// TIA Portal V18 export
// export: Created 2026-06-22T11:43:40.4217629Z, ExportSetting WithDefaults, DisplayName Totally Integrated Automation Portal, DisplayVersion V18, DisplayName TIA Portal Openness, DisplayVersion V18, DisplayName TIA Portal Version Control Interface, DisplayVersion V18, DisplayName STEP 7 Professional, DisplayVersion V18, DisplayName STEP 7 Safety, DisplayVersion V18, DisplayName WinCC Professional, DisplayVersion V18
Screen "Man Tong Quan"  1440x900, Number=3
  ScreenLayer 
    GraphicView "Graphic view_1" at 0,0 size 1440x900  Picture=Thiết kế chưa có tên (2)_1
    GraphicIOField "Graphic I/O field_9" at 430,521 size 275x288  Mode=InOutput, OnValue=1, PictureList=GL_BonChua_MucDich
      ProcessValue := HMI_Anim_BonChua1_MucDich
    GraphicIOField "Graphic I/O field_10" at 154,90 size 233x295  Mode=InOutput, OnValue=1, PictureList=GL_BonTron_MucDich
      ProcessValue := HMI_Anim_Bon1_MucDich
    GraphicIOField "Graphic I/O field_2" at 904,517 size 275x288  Mode=InOutput, OnValue=1, PictureList=GL_BonChua_MucDich
      ProcessValue := HMI_Anim_BonChua2_MucDich
    GraphicIOField "Graphic I/O field_3" at 486,90 size 233x295  Mode=InOutput, OnValue=1, PictureList=GL_BonTron_MucDich
      ProcessValue := HMI_Anim_Bon2_MucDich
    GraphicIOField "Graphic I/O field_4" at 811,89 size 233x295  Mode=InOutput, OnValue=1, PictureList=GL_BonTron_MucDich
      ProcessValue := HMI_Anim_Bon4_MucDich
    GraphicIOField "Graphic I/O field_6" at 1160,89 size 233x295  Mode=InOutput, OnValue=1, PictureList=GL_BonTron_MucDich
      ProcessValue := HMI_Anim_Bon3_MucDich
    GraphicView "Graphic view_3" at 201,61 size 11x113  Picture=Graphic_24
    GraphicIOField "Graphic I/O field_5" at 189,70 size 51x78  Mode=InOutput, OnValue=1, PictureList=GL_Van_NamDoc
      ProcessValue := V3230_Nuoc_Bon1_M
    GraphicView "Graphic view_2" at 544,60 size 11x113  Picture=Graphic_24
    GraphicIOField "Graphic I/O field_12" at 533,70 size 51x78  Mode=InOutput, OnValue=1, PictureList=GL_Van_NamDoc
      ProcessValue := V3235_Nuoc_Bon2_M
    GraphicView "Graphic view_4" at 869,59 size 11x113  Picture=Graphic_24
    GraphicIOField "Graphic I/O field_13" at 860,69 size 51x78  Mode=InOutput, OnValue=1, PictureList=GL_Van_NamDoc
      ProcessValue := V3245_Nuoc_Bon4_M
    GraphicView "Graphic view_5" at 1204,58 size 11x117  Picture=Graphic_24
    GraphicIOField "Graphic I/O field_14" at 1193,67 size 51x78  Mode=InOutput, OnValue=1, PictureList=GL_Van_NamDoc
      ProcessValue := V3240_Nuoc_Bon3_M
    GraphicView "Graphic view_6" at 229,330 size 11x172  Picture=Graphic_24
    GraphicIOField "Graphic I/O field_11" at 220,429 size 51x78  Mode=InOutput, OnValue=1, PictureList=GL_Van_NamDoc
      ProcessValue := V3233_Xa_Bon1_M
    GraphicIOField "Graphic I/O field_8" at 220,339 size 51x78  Mode=InOutput, OnValue=1, PictureList=GL_Van_NamDoc
      ProcessValue := V3232_Xa_Bon1_M
    GraphicView "Graphic view_7" at 568,331 size 11x211  Picture=Graphic_24
    GraphicView "Graphic view_8" at 869,328 size 11x164  Picture=Graphic_24
    GraphicView "Graphic view_9" at 1224,328 size 11x164  Picture=Graphic_24
    GraphicIOField "Graphic I/O field_15" at 556,341 size 51x78  Mode=InOutput, OnValue=1, PictureList=GL_Van_NamDoc
      ProcessValue := V3237_Xa_Bon2_M
    GraphicIOField "Graphic I/O field_16" at 558,417 size 51x78  Mode=InOutput, OnValue=1, PictureList=GL_Van_NamDoc
      ProcessValue := V3238_Xa_Bon2_M
    GraphicIOField "Graphic I/O field_18" at 857,346 size 51x78  Mode=InOutput, OnValue=1, PictureList=GL_Van_NamDoc
      ProcessValue := V3247_Xa_Bon4_M
    GraphicIOField "Graphic I/O field_20" at 857,412 size 51x78  Mode=InOutput, OnValue=1, PictureList=GL_Van_NamDoc
      ProcessValue := V3248_Xa_Bon4_M
    GraphicIOField "Graphic I/O field_19" at 1214,347 size 51x78  Mode=InOutput, OnValue=1, PictureList=GL_Van_NamDoc
      ProcessValue := V3242_Xa_Bon3_M
    GraphicIOField "Graphic I/O field_21" at 1213,419 size 51x78  Mode=InOutput, OnValue=1, PictureList=GL_Van_NamDoc
      ProcessValue := V3243_Xa_Bon3_M
    GraphicView "Graphic view_10" at 223,500 size 25x5  Picture=Graphic_25
    GraphicView "Graphic view_11" at 1216,490 size 25x5  Picture=Graphic_25
    GraphicView "Graphic view_12" at 223,523 size 25x5  Picture=Graphic_25
    GraphicView "Graphic view_13" at 1216,515 size 25x5  Picture=Graphic_25
    GraphicView "Graphic view_14" at 252,501 size 5x26  Picture=Graphic_24
    GraphicView "Graphic view_15" at 1206,492 size 5x26  Picture=Graphic_24
    GraphicView "Graphic view_16" at 254,510 size 242x11  Picture=Graphic_25
    GraphicView "Graphic view_17" at 487,513 size 11x57  Picture=Graphic_24
    GraphicView "Graphic view_18" at 521,159 size 11x19  Picture=Graphic_24
    GraphicView "Graphic view_19" at 440,157 size 90x11  Picture=Graphic_25
    GraphicView "Graphic view_20" at 437,160 size 11x408  Picture=Graphic_24
    GraphicView "Graphic view_21" at 231,560 size 213x11  Picture=Graphic_25
    GraphicView "Graphic view_22" at 228,525 size 11x44  Picture=Graphic_24
    GraphicView "Graphic view_23" at 630,485 size 248x11  Picture=Graphic_25
    GraphicView "Graphic view_24" at 626,488 size 11x75  Picture=Graphic_24
    GraphicView "Graphic view_25" at 640,503 size 11x68  Picture=Graphic_24
    GraphicView "Graphic view_26" at 644,501 size 566x11  Picture=Graphic_25
    GraphicView "Graphic view_27" at 1224,517 size 11x51  Picture=Graphic_24
    GraphicView "Graphic view_28" at 1142,560 size 90x11  Picture=Graphic_25
    GraphicView "Graphic view_29" at 1139,99 size 11x469  Picture=Graphic_24
    GraphicView "Graphic view_30" at 1005,93 size 143x11  Picture=Graphic_25
    GraphicView "Graphic view_31" at 1000,95 size 11x86  Picture=Graphic_24
    GraphicView "Graphic view_32" at 564,755 size 11x103  Picture=Graphic_24
    GraphicIOField "Graphic I/O field_24" at 554,759 size 51x78  Mode=InOutput, OnValue=1, PictureList=GL_Van_NamDoc
      ProcessValue := V3331_Xa_BonChua1_M
    GraphicView "Graphic view_33" at 567,849 size 22x11  Picture=Graphic_25
    GraphicView "Graphic view_34" at 581,833 size 11x40  Picture=Graphic_24
    GraphicView "Graphic view_36" at 132,426 size 8x44  Picture=Graphic_28
    GraphicView "Graphic view_35" at 133,425 size 103x6  Picture=Graphic_29
    GraphicIOField "Graphic I/O field_7" at 133,396 size 83x47  Mode=InOutput, OnValue=1, PictureList=GL_Van_NamNgang
      ProcessValue := V3234_Xa_Bon1_M
    GraphicIOField "Graphic I/O field_33" at 282,542 size 60x42  Mode=InOutput, OnValue=1, PictureList=GL_Pump_ChuyenDich
      ProcessValue := Pump3264_Chuyen_Nhanh1_M
    GraphicView "Graphic view_38" at 371,61 size 2x119  Picture=Graphic_24
    GraphicView "Graphic view_40" at 352,178 size 22x2  Picture=Graphic_25
    GraphicView "Graphic view_39" at 361,99 size 21x47  Picture=Graphic_32
    GraphicView "Graphic view_41" at 125,453 size 21x47  Picture=Graphic_32
    GraphicView "Graphic view_37" at 341,167 size 28x25  Picture=Graphic_34
    GraphicView "Graphic view_42" at 473,422 size 103x6  Picture=Graphic_29
    GraphicIOField "Graphic I/O field_17" at 471,394 size 83x47  Mode=InOutput, OnValue=1, PictureList=GL_Van_NamNgang
      ProcessValue := V3239_Xa_Bon2_M
    GraphicView "Graphic view_43" at 472,423 size 8x44  Picture=Graphic_28
    GraphicView "Graphic view_44" at 466,451 size 21x47  Picture=Graphic_32
    GraphicView "Graphic view_45" at 872,415 size 108x6  Picture=Graphic_29
    GraphicIOField "Graphic I/O field_22" at 903,387 size 83x47  Mode=InOutput, OnValue=1, PictureList=GL_Van_NamNgang
      ProcessValue := V3249_Xa_Bon4_M
    GraphicView "Graphic view_46" at 976,415 size 8x35  Picture=Graphic_28
    GraphicView "Graphic view_47" at 970,434 size 21x47  Picture=Graphic_32
    GraphicView "Graphic view_48" at 1226,422 size 118x6  Picture=Graphic_29
    GraphicIOField "Graphic I/O field_23" at 1257,394 size 83x47  Mode=InOutput, OnValue=1, PictureList=GL_Van_NamNgang
      ProcessValue := V3244_Xa_Bon3_M
    GraphicView "Graphic view_49" at 1336,422 size 8x35  Picture=Graphic_28
    GraphicView "Graphic view_50" at 1331,441 size 21x47  Picture=Graphic_32
    GraphicView "Graphic view_51" at 709,59 size 2x119  Picture=Graphic_24
    GraphicView "Graphic view_52" at 1047,60 size 2x116  Picture=Graphic_24
    GraphicView "Graphic view_53" at 1387,60 size 2x114  Picture=Graphic_24
    GraphicView "Graphic view_54" at 700,102 size 21x47  Picture=Graphic_32
    GraphicView "Graphic view_55" at 1038,104 size 21x47  Picture=Graphic_32
    GraphicView "Graphic view_56" at 1378,106 size 21x47  Picture=Graphic_32
    GraphicView "Graphic view_57" at 689,177 size 22x2  Picture=Graphic_25
    GraphicView "Graphic view_58" at 1016,175 size 33x2  Picture=Graphic_25
    GraphicView "Graphic view_59" at 1366,173 size 22x2  Picture=Graphic_25
    GraphicView "Graphic view_60" at 672,166 size 28x25  Picture=Graphic_34
    GraphicView "Graphic view_61" at 1000,165 size 28x25  Picture=Graphic_34
    GraphicView "Graphic view_62" at 1347,162 size 28x25  Picture=Graphic_34
    GraphicView "Graphic view_63" at 584,865 size 16x11  Picture=Graphic_25
    GraphicView "Graphic view_64" at 584,830 size 159x11  Picture=Graphic_25
    GraphicView "Graphic view_65" at 598,858 size 5x26  Picture=Graphic_24
    GraphicView "Graphic view_66" at 603,858 size 5x26  Picture=Graphic_24
    GraphicView "Graphic view_67" at 605,866 size 68x11  Picture=Graphic_25
    GraphicIOField "Graphic I/O field_1" at 608,851 size 60x42  Mode=InOutput, OnValue=1, PictureList=GL_Pump_ChuyenDich
      ProcessValue := Pump3362_Xa_BonChua1_M
    GraphicView "Graphic view_68" at 668,858 size 5x26  Picture=Graphic_24
    GraphicView "Graphic view_69" at 674,858 size 5x26  Picture=Graphic_24
    GraphicView "Graphic view_70" at 675,866 size 13x11  Picture=Graphic_25
    GraphicView "Graphic view_71" at 682,513 size 11x361  Picture=Graphic_24
    GraphicIOField "Graphic I/O field_25" at 672,597 size 51x78  Mode=InOutput, OnValue=1, PictureList=GL_Van_NamDoc
      ProcessValue := V3333_DieuHuong_BonChua1_M
    GraphicView "Graphic view_72" at 684,510 size 376x11  Picture=Graphic_25
    GraphicView "Graphic view_73" at 1053,512 size 11x26  Picture=Graphic_24
    GraphicIOField "Graphic I/O field_34" at 587,792 size 90x71  Mode=InOutput, OnValue=1, PictureList=GL_Pump_TuanHoanLoc
      ProcessValue := Pump3361_LuanChuyen_BonChua1_M
    GraphicView "Graphic view_74" at 735,752 size 11x144  Picture=Graphic_24
    GraphicIOField "Graphic I/O field_27" at 725,829 size 51x78  Mode=InOutput, OnValue=1, PictureList=GL_Van_NamDoc
      ProcessValue := V3335_DieuHuong_BonChua1_M
    GraphicIOField "Graphic I/O field_26" at 725,757 size 51x78  Mode=InOutput, OnValue=1, PictureList=GL_Van_NamDoc
      ProcessValue := V3334_DieuHuong_BonChua1_M
    GraphicView "Graphic view_75" at 739,889 size 528x11  Picture=Graphic_25
    GraphicView "Graphic view_76" at 738,748 size 65x11  Picture=Graphic_25
    GraphicView "Graphic view_77" at 799,521 size 11x236  Picture=Graphic_24
    GraphicView "Graphic view_78" at 801,518 size 211x11  Picture=Graphic_25
    GraphicView "Graphic view_79" at 1005,520 size 11x38  Picture=Graphic_24
    GraphicView "Graphic view_80" at 469,833 size 103x6  Picture=Graphic_29
    GraphicView "Graphic view_81" at 467,834 size 8x44  Picture=Graphic_28
    GraphicView "Graphic view_82" at 461,854 size 21x47  Picture=Graphic_32
    GraphicIOField "Graphic I/O field_30" at 467,804 size 83x47  Mode=InOutput, OnValue=1, PictureList=GL_Van_NamNgang
      ProcessValue := V3332_Xa_BonChua1_M
    GraphicView "Graphic view_83" at 1040,751 size 11x75  Picture=Graphic_24
    GraphicIOField "Graphic I/O field_28" at 1030,754 size 51x78  Mode=InOutput, OnValue=1, PictureList=GL_Van_NamDoc
      ProcessValue := V3338_Xa_BonChua2_M
    GraphicView "Graphic view_84" at 1042,818 size 62x11  Picture=Graphic_25
    GraphicView "Graphic view_85" at 1100,802 size 11x40  Picture=Graphic_24
    GraphicView "Graphic view_86" at 1104,800 size 103x11  Picture=Graphic_25
    GraphicIOField "Graphic I/O field_35" at 1108,764 size 90x71  Mode=InOutput, OnValue=1, PictureList=GL_Pump_TuanHoanLoc
      ProcessValue := Pump3364_Filter_M
    GraphicView "Graphic view_87" at 1103,833 size 12x11  Picture=Graphic_25
    GraphicView "Graphic view_88" at 1112,825 size 5x26  Picture=Graphic_24
    GraphicView "Graphic view_89" at 1117,825 size 5x26  Picture=Graphic_24
    GraphicView "Graphic view_90" at 1118,833 size 72x11  Picture=Graphic_25
    GraphicIOField "Graphic I/O field_36" at 1123,820 size 60x42  Mode=InOutput, OnValue=1, PictureList=GL_Pump_ChuyenDich
      ProcessValue := Pump3365_Filter_M
    GraphicView "Graphic view_91" at 1186,825 size 5x26  Picture=Graphic_24
    GraphicView "Graphic view_92" at 1192,825 size 5x26  Picture=Graphic_24
    GraphicView "Graphic view_93" at 1195,833 size 13x11  Picture=Graphic_25
    GraphicView "Graphic view_94" at 1201,589 size 11x252  Picture=Graphic_24
    GraphicIOField "Graphic I/O field_29" at 1191,655 size 51x78  Mode=InOutput, OnValue=1, PictureList=GL_Van_NamDoc
      ProcessValue := V3340_Duong_Filter_M
    GraphicIOField "Graphic I/O field_37" at 1156,541 size 60x42  Mode=InOutput, OnValue=1, PictureList=GL_Pump_ChuyenDich
      ProcessValue := Pump3265_Chuyen_Nhanh2_M
    GraphicView "Graphic view_95" at 1204,587 size 150x11  Picture=Graphic_25
    GraphicView "Graphic view_96" at 1257,590 size 11x307  Picture=Graphic_24
    GraphicView "Graphic view_97" at 1345,589 size 11x192  Picture=Graphic_24
    GraphicView "Graphic view_98" at 1352,589 size 75x6  Picture=Graphic_29
    GraphicIOField "Graphic I/O field_32" at 1346,558 size 83x47  Mode=InOutput, OnValue=1, PictureList=GL_Van_NamNgang
      ProcessValue := V3341_Duong_Filter_M
    GraphicView "Graphic view_99" at 1420,591 size 8x35  Picture=Graphic_28
    GraphicView "Graphic view_100" at 1414,607 size 21x47  Picture=Graphic_32
    GraphicView "Graphic view_102" at 1368,50 size 41x72  Picture=Graphic_37
    GraphicView "Graphic view_103" at 1365,159 size 28x31  Picture=Graphic_38
    GraphicView "Graphic view_104" at 1027,50 size 41x72  Picture=Graphic_37
    GraphicView "Graphic view_105" at 690,50 size 41x72  Picture=Graphic_37
    GraphicView "Graphic view_106" at 352,50 size 41x72  Picture=Graphic_37
    GraphicView "Graphic view_107" at 352,121 size 41x74  Picture=Graphic_39
    GraphicView "Graphic view_108" at 691,121 size 41x74  Picture=Graphic_39
    GraphicView "Graphic view_109" at 1028,121 size 41x74  Picture=Graphic_39
    GraphicView "Graphic view_110" at 1368,119 size 41x74  Picture=Graphic_39
    GraphicView "Graphic view_101" at 1012,165 size 45x26  Picture=Graphic_40
    GraphicView "Graphic view_111" at 676,167 size 45x26  Picture=Graphic_40
    GraphicView "Graphic view_112" at 341,167 size 38x26  Picture=Graphic_40
    GraphicIOField "Graphic I/O field_38" at 123,84 size 292x298  Mode=Output, OnValue=1, PictureList=GL_Khuay_8Frame
      ProcessValue := HMI_Anim_Bon1_Frame
    GraphicIOField "Graphic I/O field_39" at 459,83 size 292x298  Mode=InOutput, OnValue=1, PictureList=GL_Khuay_8Frame
      ProcessValue := HMI_Anim_Bon2_Frame
    GraphicIOField "Graphic I/O field_40" at 782,86 size 292x298  Mode=InOutput, OnValue=1, PictureList=GL_Khuay_8Frame
      ProcessValue := HMI_Anim_Bon4_Frame
    GraphicIOField "Graphic I/O field_41" at 1130,89 size 292x298  Mode=InOutput, OnValue=1, PictureList=GL_Khuay_8Frame
      ProcessValue := HMI_Anim_Bon3_Frame
    GraphicView "Graphic view_113" at 1280,567 size 56x45  Picture=Graphic_44
    GraphicView "Graphic view_115" at 1338,606 size 28x43  Picture=Graphic_46
    GraphicView "Graphic view_114" at 1246,722 size 28x43  Picture=Graphic_46
    GraphicView "Graphic view_116" at 1340,714 size 33x47  Picture=Graphic_47
    GraphicView "Graphic view_117" at 1327,779 size 50x52  Picture=Graphic_48
    GraphicView "Graphic view_118" at 1341,815 size 21x47  Picture=Graphic_32
    GraphicView "Graphic view_119" at 1337,843 size 29x56  Picture=Graphic_49
    GraphicView "Graphic view_120" at 939,821 size 108x6  Picture=Graphic_29
    GraphicIOField "Graphic I/O field_31" at 930,792 size 83x47  Mode=InOutput, OnValue=1, PictureList=GL_Van_NamNgang
      ProcessValue := V3339_Xa_BonChua2_M
    GraphicView "Graphic view_121" at 934,821 size 8x44  Picture=Graphic_28
    GraphicView "Graphic view_122" at 929,842 size 21x47  Picture=Graphic_32
    IOField "I/O field_1" at 113,69 size 67x32  DataFormat=Decimal, FormatPattern=999999, Mode=InOutput
    GraphicView "Graphic view_123" at 775,636 size 55x48  Picture=Graphic_50
    IOField "I/O field_2" at 300,127 size 67x28  DataFormat=Decimal, FormatPattern=999999, Mode=InOutput
    TextField "AI_Lbl_Graphic I/O field_5" at 184,48 size 60x20  StyleItem=Text field, Text="<body><p>V32.30</p></body>"
    TextField "AI_Lbl_Graphic I/O field_12" at 528,48 size 60x20  StyleItem=Text field, Text="<body><p>V32.35</p></body>"
    TextField "AI_Lbl_Graphic I/O field_13" at 855,47 size 60x20  StyleItem=Text field, Text="<body><p>V32.45</p></body>"
    TextField "AI_Lbl_Graphic I/O field_14" at 1188,45 size 60x20  StyleItem=Text field, Text="<body><p>V32.40</p></body>"
    TextField "AI_Lbl_Graphic I/O field_8" at 215,317 size 60x20  StyleItem=Text field, Text="<body><p>V32.32</p></body>"
    TextField "AI_Lbl_Graphic I/O field_11" at 215,407 size 60x20  StyleItem=Text field, Text="<body><p>V32.33</p></body>"
    TextField "AI_Lbl_Graphic I/O field_7" at 144,445 size 60x20  StyleItem=Text field, Text="<body><p>V32.34</p></body>"
    TextField "AI_Lbl_Graphic I/O field_15" at 551,319 size 60x20  StyleItem=Text field, Text="<body><p>V32.37</p></body>"
    TextField "AI_Lbl_Graphic I/O field_16" at 553,395 size 60x20  StyleItem=Text field, Text="<body><p>V32.38</p></body>"
    TextField "AI_Lbl_Graphic I/O field_17" at 482,443 size 60x20  StyleItem=Text field, Text="<body><p>V32.39</p></body>"
    TextField "AI_Lbl_Graphic I/O field_18" at 852,324 size 60x20  StyleItem=Text field, Text="<body><p>V32.47</p></body>"
    TextField "AI_Lbl_Graphic I/O field_20" at 852,390 size 60x20  StyleItem=Text field, Text="<body><p>V32.48</p></body>"
    TextField "AI_Lbl_Graphic I/O field_22" at 914,436 size 60x20  StyleItem=Text field, Text="<body><p>V32.49</p></body>"
    TextField "AI_Lbl_Graphic I/O field_19" at 1209,325 size 60x20  StyleItem=Text field, Text="<body><p>V32.42</p></body>"
    TextField "AI_Lbl_Graphic I/O field_21" at 1208,397 size 60x20  StyleItem=Text field, Text="<body><p>V32.43</p></body>"
    TextField "AI_Lbl_Graphic I/O field_23" at 1268,443 size 60x20  StyleItem=Text field, Text="<body><p>V32.44</p></body>"
    TextField "AI_Lbl_Graphic I/O field_33" at 282,586 size 60x20  StyleItem=Text field, Text="<body><p>Pump 32.64</p></body>"
    TextField "AI_Lbl_Graphic I/O field_37" at 1156,585 size 60x20  StyleItem=Text field, Text="<body><p>Pump 32.69</p></body>"
    TextField "AI_Lbl_Graphic I/O field_24" at 549,737 size 60x20  StyleItem=Text field, Text="<body><p>V33.31</p></body>"
    TextField "AI_Lbl_Graphic I/O field_30" at 478,853 size 60x20  StyleItem=Text field, Text="<body><p>V33.32</p></body>"
    TextField "AI_Lbl_Graphic I/O field_25" at 667,575 size 60x20  StyleItem=Text field, Text="<body><p>V33.33</p></body>"
    TextField "AI_Lbl_Graphic I/O field_26" at 720,735 size 60x20  StyleItem=Text field, Text="<body><p>V33.34</p></body>"
    TextField "AI_Lbl_Graphic I/O field_27" at 720,807 size 60x20  StyleItem=Text field, Text="<body><p>V33.35</p></body>"
    TextField "AI_Lbl_Graphic I/O field_34" at 602,865 size 60x20  StyleItem=Text field, Text="<body><p>Pump 33.61</p></body>"
    TextField "AI_Lbl_Graphic I/O field_1" at 676,862 size 72x20  StyleItem=Text field, Text="<body><p>Pump 33.62</p></body>"
    TextField "AI_Lbl_Graphic I/O field_28" at 1025,732 size 60x20  StyleItem=Text field, Text="<body><p>V33.38</p></body>"
    TextField "AI_Lbl_Graphic I/O field_31" at 941,841 size 60x20  StyleItem=Text field, Text="<body><p>V33.39</p></body>"
    TextField "AI_Lbl_Graphic I/O field_35" at 1123,837 size 60x20  StyleItem=Text field, Text="<body><p>Pump 33.64</p></body>"
    TextField "AI_Lbl_Graphic I/O field_36" at 1123,864 size 60x20  StyleItem=Text field, Text="<body><p>Pump 33.65</p></body>"
    TextField "AI_Lbl_Graphic I/O field_29" at 1186,633 size 60x20  StyleItem=Text field, Text="<body><p>V33.40</p></body>"
    TextField "AI_Lbl_Graphic I/O field_32" at 1357,607 size 60x20  StyleItem=Text field, Text="<body><p>V33.41</p></body>"
    IOField "AI_IO_FT3200" at 114,70 size 72x26  FormatPattern=999.9, Mode=Output, StyleItem=I/O field
      ProcessValue := FQ3200_Bon1_Eff
    TextField "AI_Lbl_AI_IO_FT3200" at 114,45 size 72x20  StyleItem=Text field, Text="<body><p>FT 32.00</p></body>"
    TextField "AI_Unit_AI_IO_FT3200" at 194,70 size 45x26  StyleItem=Text field, Text="<body><p>L</p></body>"
    IOField "AI_IO_CV3201" at 114,105 size 72x26  FormatPattern=999.9, Mode=Output, StyleItem=I/O field
      ProcessValue := CV3201_Nuoc_Bon1_M
    TextField "AI_Lbl_AI_IO_CV3201" at 114,80 size 72x20  StyleItem=Text field, Text="<body><p>CV 32.01</p></body>"
    TextField "AI_Unit_AI_IO_CV3201" at 194,105 size 45x26  StyleItem=Text field, Text="<body><p>%</p></body>"
    IOField "AI_IO_LT3203" at 300,130 size 72x26  FormatPattern=999.9, Mode=Output, StyleItem=I/O field
      ProcessValue := LT3203_Bon1_Eff
    TextField "AI_Lbl_AI_IO_LT3203" at 300,105 size 72x20  StyleItem=Text field, Text="<body><p>LT 32.03</p></body>"
    TextField "AI_Unit_AI_IO_LT3203" at 380,130 size 45x26  StyleItem=Text field, Text="<body><p>%</p></body>"
    IOField "AI_IO_TT3204" at 300,200 size 72x26  FormatPattern=99.9, Mode=Output, StyleItem=I/O field
      ProcessValue := TT3204_Bon1_Eff
    TextField "AI_Lbl_AI_IO_TT3204" at 300,175 size 72x20  StyleItem=Text field, Text="<body><p>TT 32.04</p></body>"
    TextField "AI_Unit_AI_IO_TT3204" at 380,200 size 45x26  StyleItem=Text field, Text="<body><p>°C</p></body>"
    IOField "AI_IO_FT3205" at 446,70 size 72x26  FormatPattern=999.9, Mode=Output, StyleItem=I/O field
      ProcessValue := FQ3205_Bon2_Eff
    TextField "AI_Lbl_AI_IO_FT3205" at 446,45 size 72x20  StyleItem=Text field, Text="<body><p>FT 32.05</p></body>"
    TextField "AI_Unit_AI_IO_FT3205" at 526,70 size 45x26  StyleItem=Text field, Text="<body><p>L</p></body>"
    IOField "AI_IO_CV3206" at 446,105 size 72x26  FormatPattern=999.9, Mode=Output, StyleItem=I/O field
      ProcessValue := CV3206_Hoi_Bon2_M
    TextField "AI_Lbl_AI_IO_CV3206" at 446,80 size 72x20  StyleItem=Text field, Text="<body><p>CV 32.06</p></body>"
    TextField "AI_Unit_AI_IO_CV3206" at 526,105 size 45x26  StyleItem=Text field, Text="<body><p>%</p></body>"
    IOField "AI_IO_LT3209" at 632,130 size 72x26  FormatPattern=999.9, Mode=Output, StyleItem=I/O field
      ProcessValue := LT3209_Bon2_Eff
    TextField "AI_Lbl_AI_IO_LT3209" at 632,105 size 72x20  StyleItem=Text field, Text="<body><p>LT 32.09</p></body>"
    TextField "AI_Unit_AI_IO_LT3209" at 712,130 size 45x26  StyleItem=Text field, Text="<body><p>%</p></body>"
    IOField "AI_IO_TT3208" at 632,200 size 72x26  FormatPattern=99.9, Mode=Output, StyleItem=I/O field
      ProcessValue := TT3208_Bon2_Eff
    TextField "AI_Lbl_AI_IO_TT3208" at 632,175 size 72x20  StyleItem=Text field, Text="<body><p>TT 32.08</p></body>"
    TextField "AI_Unit_AI_IO_TT3208" at 712,200 size 45x26  StyleItem=Text field, Text="<body><p>°C</p></body>"
    IOField "AI_IO_FT3215" at 771,69 size 72x26  FormatPattern=999.9, Mode=Output, StyleItem=I/O field
      ProcessValue := FQ3215_Bon4_Eff
    TextField "AI_Lbl_AI_IO_FT3215" at 771,44 size 72x20  StyleItem=Text field, Text="<body><p>FT 32.15</p></body>"
    TextField "AI_Unit_AI_IO_FT3215" at 851,69 size 45x26  StyleItem=Text field, Text="<body><p>L</p></body>"
    IOField "AI_IO_CV3216" at 771,104 size 72x26  FormatPattern=999.9, Mode=Output, StyleItem=I/O field
      ProcessValue := CV3216_Hoi_Bon4_M
    TextField "AI_Lbl_AI_IO_CV3216" at 771,79 size 72x20  StyleItem=Text field, Text="<body><p>CV 32.16</p></body>"
    TextField "AI_Unit_AI_IO_CV3216" at 851,104 size 45x26  StyleItem=Text field, Text="<body><p>%</p></body>"
    IOField "AI_IO_LT3219" at 957,129 size 72x26  FormatPattern=999.9, Mode=Output, StyleItem=I/O field
      ProcessValue := LT3218_Bon4_Eff
    TextField "AI_Lbl_AI_IO_LT3219" at 957,104 size 72x20  StyleItem=Text field, Text="<body><p>LT 32.18</p></body>"
    TextField "AI_Unit_AI_IO_LT3219" at 1037,129 size 45x26  StyleItem=Text field, Text="<body><p>%</p></body>"
    IOField "AI_IO_TT3218" at 957,199 size 72x26  FormatPattern=99.9, Mode=Output, StyleItem=I/O field
      ProcessValue := TT3219_Bon4_Eff
    TextField "AI_Lbl_AI_IO_TT3218" at 957,174 size 72x20  StyleItem=Text field, Text="<body><p>TT 32.19</p></body>"
    TextField "AI_Unit_AI_IO_TT3218" at 1037,199 size 45x26  StyleItem=Text field, Text="<body><p>°C</p></body>"
    IOField "AI_IO_FT3210" at 1120,69 size 72x26  FormatPattern=999.9, Mode=Output, StyleItem=I/O field
      ProcessValue := FQ3210_Bon3_Eff
    TextField "AI_Lbl_AI_IO_FT3210" at 1120,44 size 72x20  StyleItem=Text field, Text="<body><p>FT 32.10</p></body>"
    TextField "AI_Unit_AI_IO_FT3210" at 1200,69 size 45x26  StyleItem=Text field, Text="<body><p>L</p></body>"
    IOField "AI_IO_CV3211" at 1120,104 size 72x26  FormatPattern=999.9, Mode=Output, StyleItem=I/O field
      ProcessValue := CV3211_Nuoc_Bon3_M
    TextField "AI_Lbl_AI_IO_CV3211" at 1120,79 size 72x20  StyleItem=Text field, Text="<body><p>CV 32.11</p></body>"
    TextField "AI_Unit_AI_IO_CV3211" at 1200,104 size 45x26  StyleItem=Text field, Text="<body><p>%</p></body>"
    IOField "AI_IO_LT3214" at 1306,129 size 72x26  FormatPattern=999.9, Mode=Output, StyleItem=I/O field
      ProcessValue := LT3213_Bon3_Eff
    TextField "AI_Lbl_AI_IO_LT3214" at 1306,104 size 72x20  StyleItem=Text field, Text="<body><p>LT 32.13</p></body>"
    TextField "AI_Unit_AI_IO_LT3214" at 1386,129 size 45x26  StyleItem=Text field, Text="<body><p>%</p></body>"
    IOField "AI_IO_TT3213" at 1306,199 size 72x26  FormatPattern=99.9, Mode=Output, StyleItem=I/O field
      ProcessValue := TT3214_Bon3_Eff
    TextField "AI_Lbl_AI_IO_TT3213" at 1306,174 size 72x20  StyleItem=Text field, Text="<body><p>TT 32.14</p></body>"
    TextField "AI_Unit_AI_IO_TT3213" at 1386,199 size 45x26  StyleItem=Text field, Text="<body><p>°C</p></body>"
    IOField "AI_IO_LT3302" at 580,570 size 72x26  FormatPattern=999.9, Mode=Output, StyleItem=I/O field
      ProcessValue := LT3302_BonChua1_Eff
    TextField "AI_Lbl_AI_IO_LT3302" at 580,545 size 72x20  StyleItem=Text field, Text="<body><p>LT 33.02</p></body>"
    TextField "AI_Unit_AI_IO_LT3302" at 660,570 size 45x26  StyleItem=Text field, Text="<body><p>%</p></body>"
    IOField "AI_IO_TT3301" at 580,640 size 72x26  FormatPattern=99.9, Mode=Output, StyleItem=I/O field
      ProcessValue := TT3301_BonChua1_Eff
    TextField "AI_Lbl_AI_IO_TT3301" at 580,615 size 72x20  StyleItem=Text field, Text="<body><p>TT 33.01</p></body>"
    TextField "AI_Unit_AI_IO_TT3301" at 660,640 size 45x26  StyleItem=Text field, Text="<body><p>°C</p></body>"
    IOField "AI_IO_LT3307" at 1054,566 size 72x26  FormatPattern=999.9, Mode=Output, StyleItem=I/O field
      ProcessValue := LT3307_BonChua2_Eff
    TextField "AI_Lbl_AI_IO_LT3307" at 1054,541 size 72x20  StyleItem=Text field, Text="<body><p>LT 33.07</p></body>"
    TextField "AI_Unit_AI_IO_LT3307" at 1134,566 size 45x26  StyleItem=Text field, Text="<body><p>%</p></body>"
    IOField "AI_IO_TT3306" at 1054,636 size 72x26  FormatPattern=99.9, Mode=Output, StyleItem=I/O field
      ProcessValue := TT3306_BonChua2_Eff
    TextField "AI_Lbl_AI_IO_TT3306" at 1054,611 size 72x20  StyleItem=Text field, Text="<body><p>TT 33.06</p></body>"
    TextField "AI_Unit_AI_IO_TT3306" at 1134,636 size 45x26  StyleItem=Text field, Text="<body><p>°C</p></body>"
    IOField "AI_IO_TT3303" at 1270,636 size 72x26  FormatPattern=99.9, Mode=Output, StyleItem=I/O field
      ProcessValue := TT3303_TraoDoiNhiet_Eff
    TextField "AI_Lbl_AI_IO_TT3303" at 1270,611 size 72x20  StyleItem=Text field, Text="<body><p>TT 33.03</p></body>"
    TextField "AI_Unit_AI_IO_TT3303" at 1350,636 size 45x26  StyleItem=Text field, Text="<body><p>°C</p></body>"
    IOField "AI_IO_CV3304" at 1270,706 size 72x26  FormatPattern=999.9, Mode=Output, StyleItem=I/O field
      ProcessValue := CV3304_Nuoc_Lam_Mat_M
    TextField "AI_Lbl_AI_IO_CV3304" at 1270,681 size 72x20  StyleItem=Text field, Text="<body><p>CV 33.04</p></body>"
    TextField "AI_Unit_AI_IO_CV3304" at 1350,706 size 45x26  StyleItem=Text field, Text="<body><p>%</p></body>"
    IOField "AI_IO_PI3308" at 970,820 size 72x26  FormatPattern=99.9, Mode=Output, StyleItem=I/O field
      ProcessValue := PI3308_Truoc_Filter_Eff
    TextField "AI_Lbl_AI_IO_PI3308" at 970,795 size 72x20  StyleItem=Text field, Text="<body><p>PI 33.08</p></body>"
    TextField "AI_Unit_AI_IO_PI3308" at 1050,820 size 45x26  StyleItem=Text field, Text="<body><p>bar</p></body>"
    IOField "AI_IO_FT3309" at 1190,740 size 72x26  FormatPattern=999.9, Mode=Output, StyleItem=I/O field
      ProcessValue := FT3309_Xa_Thanh_Pham_Eff
    TextField "AI_Lbl_AI_IO_FT3309" at 1190,715 size 72x20  StyleItem=Text field, Text="<body><p>FT 33.09</p></body>"
    TextField "AI_Unit_AI_IO_FT3309" at 1270,740 size 45x26  StyleItem=Text field, Text="<body><p>L/h</p></body>"
    IOField "AI_IO_CVFiller" at 1290,820 size 72x26  FormatPattern=999.9, Mode=Output, StyleItem=I/O field
      ProcessValue := CV_Filler_Cap_Dich_M
    TextField "AI_Lbl_AI_IO_CVFiller" at 1290,795 size 72x20  StyleItem=Text field, Text="<body><p>CV Filler</p></body>"
    TextField "AI_Unit_AI_IO_CVFiller" at 1370,820 size 45x26  StyleItem=Text field, Text="<body><p>%</p></body>"
  SoftKey "Softkey_F5"  KeyCode=202
